// TIA Portal V17 export
// export: Created 2024-06-14T09:52:57.8468403Z, ExportSetting WithDefaults, DisplayName Totally Integrated Automation Portal, DisplayVersion V17, DisplayName TIA Portal Openness, DisplayVersion V17, DisplayName TIA Portal Version Control Interface, DisplayVersion V17, DisplayName Simotion SCOUT TIA, DisplayVersion 5.4.3.0, DisplayName SINAMICS Startdrive Advanced, DisplayVersion V17 SP1 Update 1, DisplayName SINAMICS Startdrive G110M, G120, G120C, G120D, G120P, G115D, DisplayVersion V17 SP1 Update 1, DisplayName SINAMICS Startdrive G130, G150, S120, S150, SINAMICS MV, S210, DisplayVersion V17 SP1 Update 1, DisplayName STEP 7 Professional, DisplayVersion V17, DisplayName STEP 7 Safety, DisplayVersion V17, DisplayName WinCC Professional, DisplayVersion V17
FUNCTION "Common_Logoc" : Void   // FC1, LAD
{ S7_Optimized_Access := 'TRUE' }
VERSION : 0.1
// stored: AutoNumber true, IsIECCheckEnabled false, SetENOAutomatically false, UDAEnableTagReadback false
BEGIN

REGION Network 1: Empty Network
   // Ohm Namashivaya
END_REGION

REGION Network 2: Total Enabled Stations
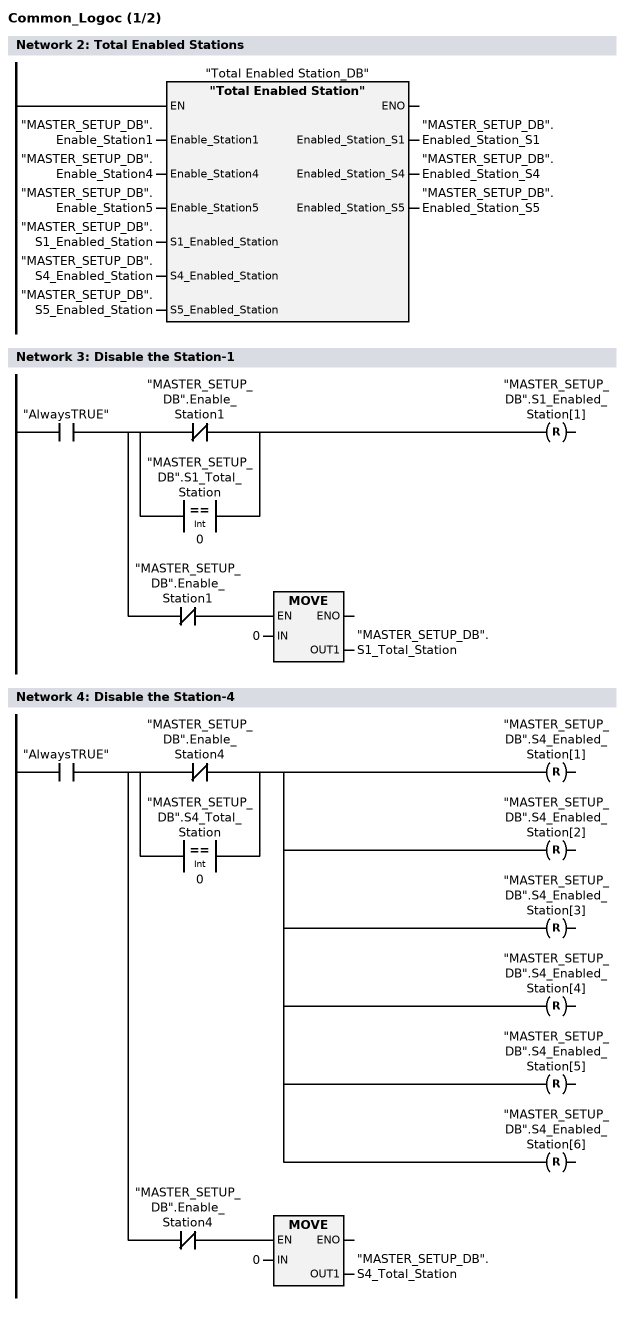
   RUNG wire#powerrail
      "Total Enabled Station_DB"(Enable_Station1 := "MASTER_SETUP_DB".Enable_Station1, Enable_Station4 := "MASTER_SETUP_DB".Enable_Station4, Enable_Station5 := "MASTER_SETUP_DB".Enable_Station5, S1_Enabled_Station := "MASTER_SETUP_DB".S1_Enabled_Station, S4_Enabled_Station := "MASTER_SETUP_DB".S4_Enabled_Station, S5_Enabled_Station := "MASTER_SETUP_DB".S5_Enabled_Station, Enabled_Station_S1 => "MASTER_SETUP_DB".Enabled_Station_S1, Enabled_Station_S4 => "MASTER_SETUP_DB".Enabled_Station_S4, Enabled_Station_S5 => "MASTER_SETUP_DB".Enabled_Station_S5)
   END_RUNG
   // the same network as SCL:
   "Total Enabled Station_DB"(Enable_Station1 := "MASTER_SETUP_DB".Enable_Station1,   // "Total Enabled Station"
                           Enable_Station4 := "MASTER_SETUP_DB".Enable_Station4,
                           Enable_Station5 := "MASTER_SETUP_DB".Enable_Station5,
                           S1_Enabled_Station := "MASTER_SETUP_DB".S1_Enabled_Station,
                           S4_Enabled_Station := "MASTER_SETUP_DB".S4_Enabled_Station,
                           S5_Enabled_Station := "MASTER_SETUP_DB".S5_Enabled_Station,
                           Enabled_Station_S1 => "MASTER_SETUP_DB".Enabled_Station_S1,
                           Enabled_Station_S4 => "MASTER_SETUP_DB".Enabled_Station_S4,
                           Enabled_Station_S5 => "MASTER_SETUP_DB".Enabled_Station_S5);
END_REGION

REGION Network 3: Disable the Station-1
   RUNG wire#powerrail
      Contact( "AlwaysTRUE" )
      wire#w1
      I_Contact( "MASTER_SETUP_DB".Enable_Station1 )
      wire#w2
      R_Coil( "MASTER_SETUP_DB".S1_Enabled_Station[1] )
   END_RUNG
   RUNG wire#w1
      { S7_Templates := "SrcType := Int" } EQ_Contact(in1 := "MASTER_SETUP_DB".S1_Total_Station, in2 := 0)
   END_RUNG wire#w2
   RUNG wire#w1
      I_Contact( "MASTER_SETUP_DB".Enable_Station1 )
      Move(in := 0, out1 => "MASTER_SETUP_DB".S1_Total_Station)
   END_RUNG
   // the same network as SCL:
   IF "AlwaysTRUE" AND (NOT "MASTER_SETUP_DB".Enable_Station1 OR ("MASTER_SETUP_DB".S1_Total_Station = 0)) THEN
       "MASTER_SETUP_DB".S1_Enabled_Station[1] := FALSE;
   END_IF;
   IF "AlwaysTRUE" AND NOT "MASTER_SETUP_DB".Enable_Station1 THEN
       "MASTER_SETUP_DB".S1_Total_Station := 0;
   END_IF;
END_REGION

REGION Network 4: Disable the Station-4
   RUNG wire#powerrail
      Contact( "AlwaysTRUE" )
      wire#w1
      I_Contact( "MASTER_SETUP_DB".Enable_Station4 )
      wire#w2
      R_Coil( "MASTER_SETUP_DB".S4_Enabled_Station[1] )
   END_RUNG
   RUNG wire#w1
      { S7_Templates := "SrcType := Int" } EQ_Contact(in1 := "MASTER_SETUP_DB".S4_Total_Station, in2 := 0)
   END_RUNG wire#w2
   RUNG wire#w2
      R_Coil( "MASTER_SETUP_DB".S4_Enabled_Station[2] )
   END_RUNG
   RUNG wire#w2
      R_Coil( "MASTER_SETUP_DB".S4_Enabled_Station[3] )
   END_RUNG
   RUNG wire#w2
      R_Coil( "MASTER_SETUP_DB".S4_Enabled_Station[4] )
   END_RUNG
   RUNG wire#w2
      R_Coil( "MASTER_SETUP_DB".S4_Enabled_Station[5] )
   END_RUNG
   RUNG wire#w2
      R_Coil( "MASTER_SETUP_DB".S4_Enabled_Station[6] )
   END_RUNG
   RUNG wire#w1
      I_Contact( "MASTER_SETUP_DB".Enable_Station4 )
      Move(in := 0, out1 => "MASTER_SETUP_DB".S4_Total_Station)
   END_RUNG
   // the same network as SCL:
   IF "AlwaysTRUE" AND (NOT "MASTER_SETUP_DB".Enable_Station4 OR ("MASTER_SETUP_DB".S4_Total_Station = 0)) THEN
       "MASTER_SETUP_DB".S4_Enabled_Station[1] := FALSE;
       "MASTER_SETUP_DB".S4_Enabled_Station[2] := FALSE;
       "MASTER_SETUP_DB".S4_Enabled_Station[3] := FALSE;
       "MASTER_SETUP_DB".S4_Enabled_Station[4] := FALSE;
       "MASTER_SETUP_DB".S4_Enabled_Station[5] := FALSE;
       "MASTER_SETUP_DB".S4_Enabled_Station[6] := FALSE;
   END_IF;
   IF "AlwaysTRUE" AND NOT "MASTER_SETUP_DB".Enable_Station4 THEN
       "MASTER_SETUP_DB".S4_Total_Station := 0;
   END_IF;
END_REGION

REGION Network 5: Disable the Station-5
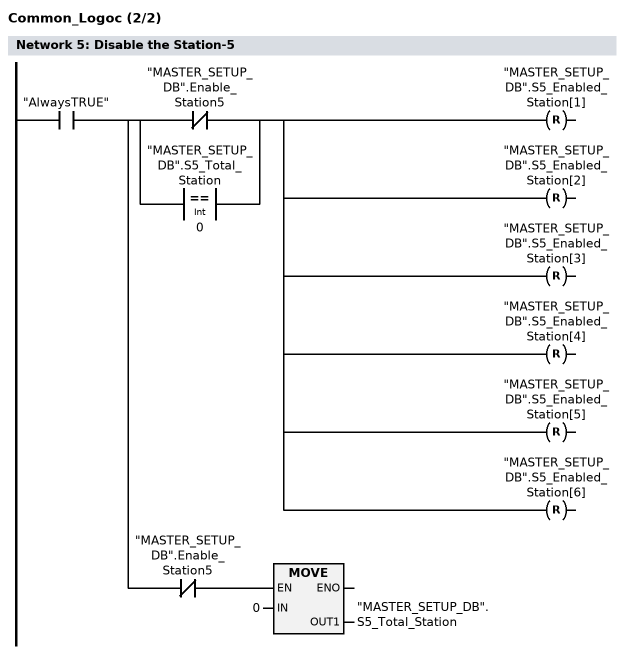
   RUNG wire#powerrail
      Contact( "AlwaysTRUE" )
      wire#w1
      I_Contact( "MASTER_SETUP_DB".Enable_Station5 )
      wire#w2
      R_Coil( "MASTER_SETUP_DB".S5_Enabled_Station[1] )
   END_RUNG
   RUNG wire#w1
      { S7_Templates := "SrcType := Int" } EQ_Contact(in1 := "MASTER_SETUP_DB".S5_Total_Station, in2 := 0)
   END_RUNG wire#w2
   RUNG wire#w2
      R_Coil( "MASTER_SETUP_DB".S5_Enabled_Station[2] )
   END_RUNG
   RUNG wire#w2
      R_Coil( "MASTER_SETUP_DB".S5_Enabled_Station[3] )
   END_RUNG
   RUNG wire#w2
      R_Coil( "MASTER_SETUP_DB".S5_Enabled_Station[4] )
   END_RUNG
   RUNG wire#w2
      R_Coil( "MASTER_SETUP_DB".S5_Enabled_Station[5] )
   END_RUNG
   RUNG wire#w2
      R_Coil( "MASTER_SETUP_DB".S5_Enabled_Station[6] )
   END_RUNG
   RUNG wire#w1
      I_Contact( "MASTER_SETUP_DB".Enable_Station5 )
      Move(in := 0, out1 => "MASTER_SETUP_DB".S5_Total_Station)
   END_RUNG
   // the same network as SCL:
   IF "AlwaysTRUE" AND (NOT "MASTER_SETUP_DB".Enable_Station5 OR ("MASTER_SETUP_DB".S5_Total_Station = 0)) THEN
       "MASTER_SETUP_DB".S5_Enabled_Station[1] := FALSE;
       "MASTER_SETUP_DB".S5_Enabled_Station[2] := FALSE;
       "MASTER_SETUP_DB".S5_Enabled_Station[3] := FALSE;
       "MASTER_SETUP_DB".S5_Enabled_Station[4] := FALSE;
       "MASTER_SETUP_DB".S5_Enabled_Station[5] := FALSE;
       "MASTER_SETUP_DB".S5_Enabled_Station[6] := FALSE;
   END_IF;
   IF "AlwaysTRUE" AND NOT "MASTER_SETUP_DB".Enable_Station5 THEN
       "MASTER_SETUP_DB".S5_Total_Station := 0;
   END_IF;
END_REGION
END_FUNCTION
